(* CoDeSys 2.3 export: SYSTEMINIT.EXP *)

(* POU SystemInit, ST *)
FUNCTION SystemInit : BOOL
(*
	Инициализация программы
	Вызывается один раз при старте ПЛК
*)
VAR_INPUT
END_VAR
VAR
END_VAR
MB_W_01 := K14UZSPumpSpeed;
(*
	Инициализация модбас параметра,
	отвечающего за сигнал на UZ
*)
END_FUNCTION
